% RSLogix 500 project I2P-JOB-23 DUNCAN_SUTTON.RSS, saved by version 10.00.00.00 %
PROJECT "ML01A"    % processor: Bul.1763 MicroLogix 1100 Series B %

PROGRAM FILES
  LAD 2   15 rungs

DATA FILES
  O0 OUTPUT  4 elements
  I1 INPUT  6 elements
  S2 STATUS  66 elements
  B3 BINARY  1 elements
  T4 TIMER  2 elements
  C5 COUNTER  2 elements
  R6 CONTROL  1 elements
  N7 INTEGER  1 elements
  F8 FLOAT  1 elements

LADDER 2
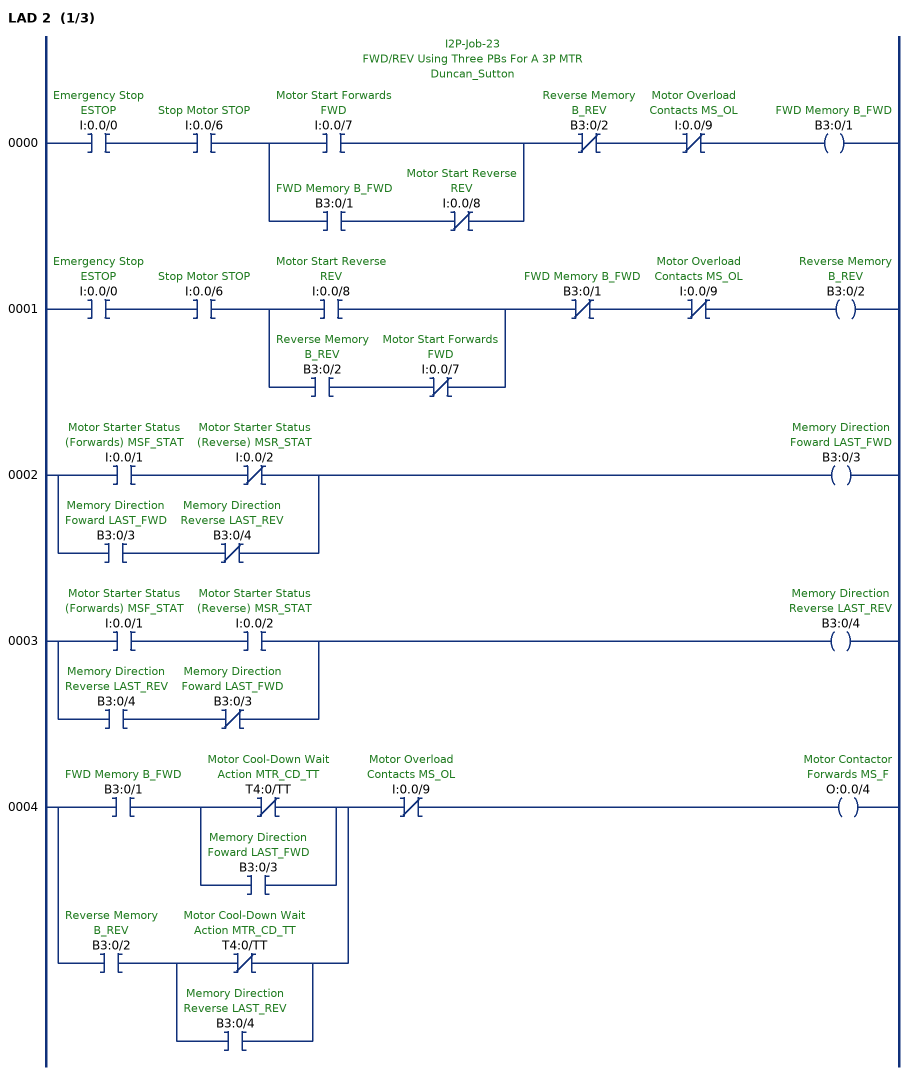
% Rung: 0 %
% I2P-Job-23
% FWD/REV Using Three PBs For A 3P MTR
% Duncan_Sutton %
SOR XIC I:0.0/0 XIC I:0.0/6 BST XIC I:0.0/7 NXB XIC B3:0/1 XIO I:0.0/8 BND XIO B3:0/2 XIO I:0.0/9 OTE B3:0/1 EOR
%   I:0.0/0  ESTOP  "Emergency Stop" %
%   I:0.0/6  STOP  "Stop Motor" %
%   I:0.0/7  FWD  "Motor Start Forwards" %
%   B3:0/1  B_FWD  "FWD Memory" %
%   I:0.0/8  REV  "Motor Start Reverse" %
%   B3:0/2  B_REV  "Reverse Memory" %
%   I:0.0/9  MS_OL  "Motor Overload Contacts" %
% Rung: 1 %
SOR XIC I:0.0/0 XIC I:0.0/6 BST XIC I:0.0/8 NXB XIC B3:0/2 XIO I:0.0/7 BND XIO B3:0/1 XIO I:0.0/9 OTE B3:0/2 EOR
%   I:0.0/0  ESTOP  "Emergency Stop" %
%   I:0.0/6  STOP  "Stop Motor" %
%   I:0.0/8  REV  "Motor Start Reverse" %
%   B3:0/2  B_REV  "Reverse Memory" %
%   I:0.0/7  FWD  "Motor Start Forwards" %
%   B3:0/1  B_FWD  "FWD Memory" %
%   I:0.0/9  MS_OL  "Motor Overload Contacts" %
% Rung: 2 %
SOR BST XIC I:0.0/1 XIO I:0.0/2 NXB XIC B3:0/3 XIO B3:0/4 BND OTE B3:0/3 EOR
%   I:0.0/1  MSF_STAT  "Motor Starter Status (Forwards)" %
%   I:0.0/2  MSR_STAT  "Motor Starter Status (Reverse)" %
%   B3:0/3  LAST_FWD  "Memory Direction Foward" %
%   B3:0/4  LAST_REV  "Memory Direction Reverse" %
% Rung: 3 %
SOR BST XIC I:0.0/1 XIC I:0.0/2 NXB XIC B3:0/4 XIO B3:0/3 BND OTE B3:0/4 EOR
%   I:0.0/1  MSF_STAT  "Motor Starter Status (Forwards)" %
%   I:0.0/2  MSR_STAT  "Motor Starter Status (Reverse)" %
%   B3:0/4  LAST_REV  "Memory Direction Reverse" %
%   B3:0/3  LAST_FWD  "Memory Direction Foward" %
% Rung: 4 %
SOR BST XIC B3:0/1 BST XIO T4:0/TT NXB XIC B3:0/3 BND NXB XIC B3:0/2 BST XIO T4:0/TT NXB XIC B3:0/4 BND BND XIO I:0.0/9 OTE O:0.0/4 EOR
%   B3:0/1  B_FWD  "FWD Memory" %
%   T4:0/TT  MTR_CD_TT  "Motor Cool-Down Wait Action" %
%   B3:0/3  LAST_FWD  "Memory Direction Foward" %
%   B3:0/2  B_REV  "Reverse Memory" %
%   B3:0/4  LAST_REV  "Memory Direction Reverse" %
%   I:0.0/9  MS_OL  "Motor Overload Contacts" %
%   O:0.0/4  MS_F  "Motor Contactor Forwards" %

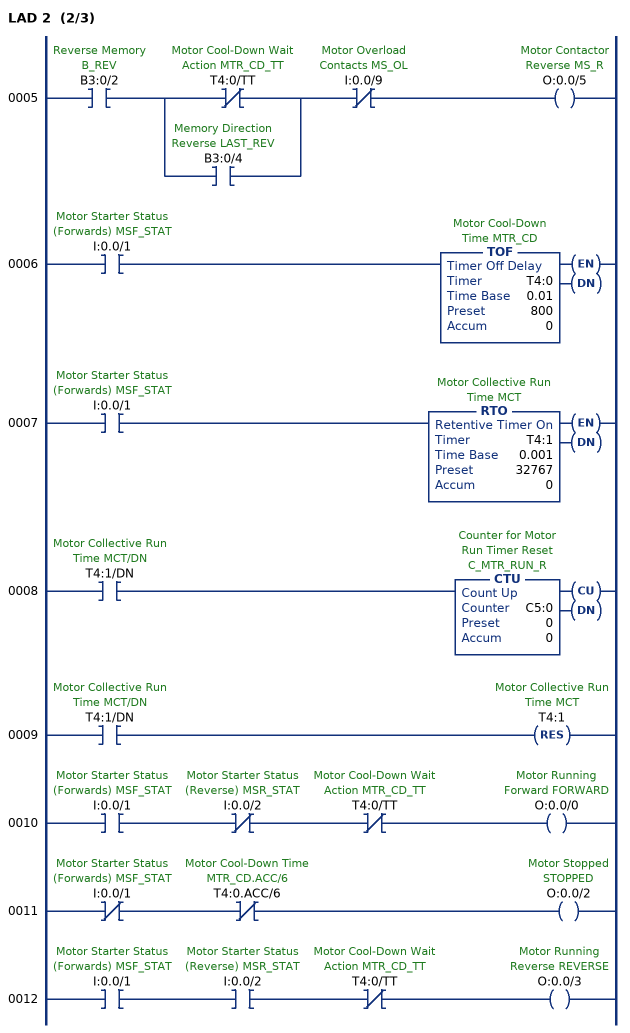
% Rung: 5 %
SOR XIC B3:0/2 BST XIO T4:0/TT NXB XIC B3:0/4 BND XIO I:0.0/9 OTE O:0.0/5 EOR
%   B3:0/2  B_REV  "Reverse Memory" %
%   T4:0/TT  MTR_CD_TT  "Motor Cool-Down Wait Action" %
%   B3:0/4  LAST_REV  "Memory Direction Reverse" %
%   I:0.0/9  MS_OL  "Motor Overload Contacts" %
%   O:0.0/5  MS_R  "Motor Contactor Reverse" %
% Rung: 6 %
SOR XIC I:0.0/1 TOF T4:0 0.01 800 0 EOR
%   I:0.0/1  MSF_STAT  "Motor Starter Status (Forwards)" %
%   T4:0  MTR_CD  "Motor Cool-Down Time" %
% Rung: 7 %
SOR XIC I:0.0/1 RTO T4:1 0.001 32767 0 EOR
%   I:0.0/1  MSF_STAT  "Motor Starter Status (Forwards)" %
%   T4:1  MCT  "Motor Collective Run Time" %
% Rung: 8 %
SOR XIC T4:1/DN CTU C5:0 0 0 EOR
%   T4:1  MCT  "Motor Collective Run Time" %
%   C5:0  C_MTR_RUN_R  "Counter for Motor Run Timer Reset" %
% Rung: 9 %
SOR XIC T4:1/DN RES T4:1 EOR
%   T4:1  MCT  "Motor Collective Run Time" %
% Rung: 10 %
SOR XIC I:0.0/1 XIO I:0.0/2 XIO T4:0/TT OTE O:0.0/0 EOR
%   I:0.0/1  MSF_STAT  "Motor Starter Status (Forwards)" %
%   I:0.0/2  MSR_STAT  "Motor Starter Status (Reverse)" %
%   T4:0/TT  MTR_CD_TT  "Motor Cool-Down Wait Action" %
%   O:0.0/0  FORWARD  "Motor Running Forward" %
% Rung: 11 %
SOR XIO I:0.0/1 XIO T4:0.ACC/6 OTE O:0.0/2 EOR
%   I:0.0/1  MSF_STAT  "Motor Starter Status (Forwards)" %
%   T4:0  MTR_CD  "Motor Cool-Down Time" %
%   O:0.0/2  STOPPED  "Motor Stopped" %
% Rung: 12 %
SOR XIC I:0.0/1 XIC I:0.0/2 XIO T4:0/TT OTE O:0.0/3 EOR
%   I:0.0/1  MSF_STAT  "Motor Starter Status (Forwards)" %
%   I:0.0/2  MSR_STAT  "Motor Starter Status (Reverse)" %
%   T4:0/TT  MTR_CD_TT  "Motor Cool-Down Wait Action" %
%   O:0.0/3  REVERSE  "Motor Running Reverse" %

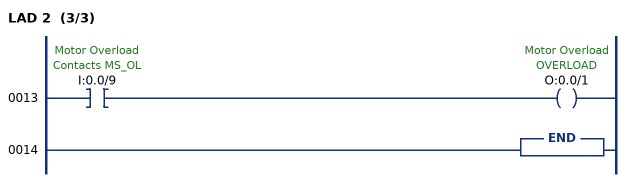
% Rung: 13 %
SOR XIC I:0.0/9 OTE O:0.0/1 EOR
%   I:0.0/9  MS_OL  "Motor Overload Contacts" %
%   O:0.0/1  OVERLOAD  "Motor Overload" %
% Rung: 14 %
SOR END EOR

OTHER DOCUMENTED ADDRESSES
  B3:0/0  B_ESTOP  "B_Estop"
  C5:1  C_MTR_T  "Collective Motor Run Time Counter"
  I:0.0/3  MODE_ON  "Valve Mode ON"
  I:0.0/4  MODE_AUTO  "Valve Mode Auto"
  I:0.0/5  MODE  "Mode: A=Run B=Jog"
  I:0.1  MS
  T4:0.ACC  MTR_CD_S  "Motor Cool-Down Time Signal"
  T4:0.ACC/0  T4
  T4:0.PRE  OVERCLOCK  "Collective Motor OverClock"
  T4:0/DN  CMT_DN  "Collective Motor Run Time Done"

DATA TABLE (non-zero values as saved)
DATA B3
% B3:0 % 0X0009
DATA T4
% .PRE .ACC %
% T4:0 % 800 0
% T4:1 % 32767 0
